// TwinCAT 3 PLC project TimerPractice
// ProgramVersion: 3.1.4022.4
// libraries:
//   Tc2_Standard, * (Beckhoff Automation GmbH)
//   Tc2_System, * (Beckhoff Automation GmbH)
//   Tc3_Module, * (Beckhoff Automation GmbH)
// project tree:
//   FBs/ FB_Timer.TcPOU (not stored)
//   GVLs/ GVL_General.TcGVL
//   / PlcTask.TcTTO
//   POUs/ MAIN.TcPOU
// real-time tasks:
//   TASK PlcTask: cycle T#10ms, priority 20, ADS port 350

CONFIGURATION TimerPractice
    RESOURCE PLC ON TwinCAT3
        TASK PlcTask(INTERVAL := T#10ms, PRIORITY := 20);
        PROGRAM MAIN WITH PlcTask : MAIN;
    END_RESOURCE
END_CONFIGURATION

// ---- GVLs/GVL_General.TcGVL
{attribute 'qualified_only'}
VAR_GLOBAL
	myTimer		:FB_Timer;
END_VAR

// ---- POUs/MAIN.TcPOU
PROGRAM MAIN
VAR
	bFlag			:BOOL;
END_VAR

GVL_General.myTimer.Delay(in:=T#5S);

IF	GVL_General.myTimer.bDone THEN 
	bFlag := TRUE;
	
	
END_IF

END_PROGRAM
